# EPICS substitutions: ek9000App/Db/EL3124.substitutions
file EL3124.template
{       pattern
        {
                TERMINAL,

        }
        {
        }
}
